FUNCTION_BLOCK FB_SRAlarmArg EXTENDS FB_SRAlarm
VAR_INPUT
    arg1		: ST_Arg;
    arg2		: ST_Arg;
	arg3		: ST_Arg;
	arg4		: ST_Arg;
	arg5		: ST_Arg;
END_VAR
VAR
	aArgStack			: ARRAY[1..ALARM_ARG_STACK_SIZE] OF BYTE;
	fbWritableArgStack	: FB_WrArgStack(ADR(aArgStack), ALARM_ARG_STACK_SIZE);
END_VAR

SUPER^();

PROPERTY ArgStackMemoryPointer : POINTER TO BYTE
GET
ArgStackMemoryPointer := fbWritableArgStack.MemoryPointer;
END_GET
END_PROPERTY

PROPERTY ArgStackMemorySize : DINT
GET
ArgStackMemorySize := fbWritableArgStack.MemorySize;
END_GET
END_PROPERTY

METHOD PROTECTED  ClearArgStack
VAR_INPUT
END_VAR
fbWritableArgStack.Clear();
END_METHOD

METHOD PROTECTED CopyArgsToStack
VAR_INPUT
END_VAR
fbWritableArgStack.AddArg(arg1);
fbWritableArgStack.AddArg(arg2);
fbWritableArgStack.AddArg(arg3);
fbWritableArgStack.AddArg(arg4);
fbWritableArgStack.AddArg(arg5);
END_METHOD

END_FUNCTION_BLOCK

(* stored: Version 1.1.0.1, ProductVersion 3.1.4024.15
   POU FB_SRAlarmArg: Id {d3030c0a-36e2-424e-a0fb-40956012db8c}, SpecialFunc None
   Property ArgStackMemoryPointer: Id {46cd283c-2405-40bb-aee3-1cc3aa092b37}
   Get Get: Id {dc1e9a1a-922e-4b9c-8eb5-12ac346ccae3}
   Property ArgStackMemorySize: Id {fccf0028-91bd-4b24-9234-390cf7c2d8e4}
   Get Get: Id {6ae3f2bb-3206-4016-8b10-5af5d273bcad}
   Method ClearArgStack: Id {3c1cd89e-a3af-4573-8c16-360c7d000724}
   Method CopyArgsToStack: Id {ce5ef490-0ad7-4008-9974-8150973bd8e1} *)
